FUNCTION_BLOCK _TcVnSize2_REAL_TestSuite EXTENDS TcUnit.FB_TestSuite
VAR
END_VAR

TestAddress();
TestClearReference();
TestClone();
TestTypeNameReturnsExpected();
TestIdentifierReturnsExpected();
//TestMakeReferenceToFollowsReference();
//TestMakeReferenceToUpdatesReference();
TestSize();
TestValueReturnsExpectedAfterInit();
TestValueReturnsExpectedAfterChange();
//TestSerializeTypeWith();
TestSerializeWith();
//TestTryDeserializeFrom();
//TestTryMakeReferenceToFollowsReference();
//TestTryMakeReferenceToUpdatesReference();

METHOD PUBLIC TestAddress
VAR
    _type : _TcVnSize2_REAL;
    notExpected : PVOID := 0;
    actual : PVOID;
END_VAR
TEST('TestAddress');

actual := _type.Address;

AssertFalse(
    Condition := (notExpected = actual),
    Message := 'Type did not return a valid address.'
);

TEST_FINISHED();
END_METHOD

METHOD PUBLIC TestClearReference
VAR
    _type : _ETcVn2dCodeSearchStrategy(ETcVn2dCodeSearchStrategy.TCVN_CSS_DEFAULT);
	target : ETcVn2dCodeSearchStrategy := ETcVn2dCodeSearchStrategy.TCVN_CSS_DEFAULT;
    expected : ETcVn2dCodeSearchStrategy := ETcVn2dCodeSearchStrategy.TCVN_CSS_DEFAULT;
    actual : ETcVn2dCodeSearchStrategy;
END_VAR
TEST('TestClearReference');

_type.MakeReferenceTo(target);
_type.ClearReference();
target := ETcVn2dCodeSearchStrategy.TCVN_CSS_FIRST_FLIPPED;

actual := _type.Value;

AssertEquals(
    Expected := expected,
    Actual := actual,
    Message := 'Value continued to follow target.'
);

TEST_FINISHED();
END_METHOD

METHOD PUBLIC TestClone
VAR
    _type : _TcVnSize2_REAL;
	clone : I_Datatype;
	isValidClone : BOOL;
	compareResult : DINT;
END_VAR
TEST('TestClone');

clone := _type.Clone();

isValidClone := clone <> 0;

IF isValidClone THEN
	compareResult := memcmp(_type.Address, clone.Address, clone.Size);
END_IF

AssertTrue(
	Condition := isValidClone,
	Message := 'Clone did not produce a clone'
);

AssertEquals_DINT(
	Expected := 0,
    Actual := compareResult,
    Message := 'Clone did not return a valid clone.'
);

clone.Dispose();

TEST_FINISHED();
END_METHOD

METHOD PUBLIC TestIdentifierReturnsExpected
VAR
    _type : _TcVnSize2_REAL;
    expected : STRING := 'TcVnSize2_REAL';
    actual : STRING;
END_VAR
TEST('TestIdentifierReturnsExpected');

actual := _type.Identifier;

AssertEquals_STRING(
    Expected := expected,
    Actual := actual,
    Message := 'Type did not return correct iec type.'
);

TEST_FINISHED();
END_METHOD

METHOD PUBLIC TestMakeReferenceToFollowsReference
VAR
    _type : _TcVnSize2_REAL;
	target : TcVnSize2_REAL;
    expected : TcVnSize2_REAL := (fWidth := 1.23, fHeight := 4.56);
    actual : TcVnSize2_REAL;
END_VAR
TEST('TestMakeReferenceToFollowsReference');

_type.MakeReferenceTo(target);
target.fWidth := 1.23;
target.fHeight := 4.56;

actual := _type.Value;

AssertEquals(
    Expected := expected,
    Actual := actual,
    Message := 'Value did not follow target change.'
);

TEST_FINISHED();
END_METHOD

METHOD PUBLIC TestMakeReferenceToUpdatesReference
VAR
    _type : _ETcVn2dCodeSearchStrategy(ETcVn2dCodeSearchStrategy.TCVN_CSS_DEFAULT);
	target : ETcVn2dCodeSearchStrategy := ETcVn2dCodeSearchStrategy.TCVN_CSS_DEFAULT;
    expected : ETcVn2dCodeSearchStrategy := ETcVn2dCodeSearchStrategy.TCVN_CSS_FIRST_FLIPPED;
    actual : ETcVn2dCodeSearchStrategy;
END_VAR
TEST('TestMakeReferenceToUpdatesReference');

_type.MakeReferenceTo(target);
_type.Value := ETcVn2dCodeSearchStrategy.TCVN_CSS_FIRST_FLIPPED;

actual := target;

AssertEquals(
    Expected := expected,
    Actual := actual,
    Message := 'Value did not update target.'
);

TEST_FINISHED();
END_METHOD

METHOD PUBLIC TestSerializeTypeWith
VAR
    _type : _TcVnSize2_REAL;
    serializer : JsonSerializer;
    //expected : STRING(500) := '{"typeName":"STRUCT","identifier":"TcVnSize2_REAL","members":{"fWidth":{"typeName":"REAL","minValue":-3.4028230607370967e38,"maxValue":3.4028230607370967      }';
    expected : STRING(500) := '';
    actual : STRING(500);
END_VAR
TEST('TestSerializeTypeWith');

serializer.Reset();
_type.SerializeTypeWith(serializer);
serializer.TryGetSerializedData(ADR(actual), SIZEOF(actual));

AssertEquals_STRING(
    Expected := expected,
    Actual := actual,
    Message := 'Serialization of type did not return correct string.'
);

TEST_FINISHED();
END_METHOD

METHOD PUBLIC TestSerializeWith
VAR
    _type : _TcVnSize2_REAL;
    serializer : JsonSerializer;
    expected : STRING := '{"fWidth":0.0,"fHeight":0.0}';
    actual : STRING(500);
END_VAR
TEST('TestSerializeWith');

serializer.Reset();
_type.SerializeWith(serializer);
serializer.TryGetSerializedData(ADR(actual), SIZEOF(actual));

AssertEquals_STRING(
    Expected := expected,
    Actual := actual,
    Message := 'Serialization of type data did not return correct string.'
);

TEST_FINISHED();
END_METHOD

METHOD PUBLIC TestSize
VAR
    _type : _TcVnSize2_REAL;
    expected : UDINT := SIZEOF(TcVnSize2_REAL);
    actual : UDINT;
END_VAR
TEST('TestSize');

actual := _type.Size;

AssertEquals_UDINT(
    Expected := Expected,
    Actual := actual,
    Message := 'Type did not return the correct size.'
);

TEST_FINISHED();
END_METHOD

METHOD PUBLIC TestTryDeserializeFrom
VAR
    deserializer : JsonDeserializer;
    feedback : DeserializerFeedback;
    json : STRING := '"TCVN_CSS_DEFAULT"';
    _type : _ETcVn2dCodeSearchStrategy(ETcVn2dCodeSearchStrategy.TCVN_CSS_DEFAULT);
    expected : ETcVn2dCodeSearchStrategy := ETcVn2dCodeSearchStrategy.TCVN_CSS_DEFAULT;
    actual : ETcVn2dCodeSearchStrategy;
 END_VAR
TEST('TestTryDeserializeFrom');

deserializer.Reset();
deserializer.TryLoad(json);
_type.TryDeserializeFrom(Deserializer, Feedback);

actual := _type.Value;

AssertEquals(
    Expected := expected,
    Actual := actual,
    Message := 'Type did not deserialize correctly.'
);

TEST_FINISHED();
END_METHOD

METHOD PUBLIC TestTryMakeReferenceToFollowsReference
VAR
    _type : _TcVnSize2_REAL;
	target : _TcVnSize2_REAL;
    expected : TcVnSize2_REAL := (fWidth := 1.23, fHeight := 4.56);
    actual : TcVnSize2_REAL;
END_VAR
TEST('TestTryMakeReferenceToFollowsReference');

_type.TryMakeReferenceTo(target);
target.Value.fHeight := 1.23;
target.Value.fHeight := 4.56;

actual := _type.Value;

AssertEquals(
    Expected := expected,
    Actual := actual,
    Message := 'Value did not follow target change.'
);

TEST_FINISHED();
END_METHOD

METHOD PUBLIC TestTryMakeReferenceToUpdatesReference
VAR
    _type : _ETcVn2dCodeSearchStrategy(ETcVn2dCodeSearchStrategy.TCVN_CSS_DEFAULT);
	target : _ETcVn2dCodeSearchStrategy(ETcVn2dCodeSearchStrategy.TCVN_CSS_DEFAULT);
    expected : ETcVn2dCodeSearchStrategy := ETcVn2dCodeSearchStrategy.TCVN_CSS_FIRST_FLIPPED;
    actual : ETcVn2dCodeSearchStrategy;
END_VAR
TEST('TestTryMakeReferenceToUpdatesReference');

_type.TryMakeReferenceTo(target);
_type.Value := ETcVn2dCodeSearchStrategy.TCVN_CSS_FIRST_FLIPPED;

actual := target.Value;

AssertEquals(
    Expected := expected,
    Actual := actual,
    Message := 'Value did not update target.'
);

TEST_FINISHED();
END_METHOD

METHOD PUBLIC TestTypeNameReturnsExpected
VAR
    _type : _TcVnSize2_REAL;
    expected : STRING := 'STRUCT';
    actual : STRING;
END_VAR
TEST('TestTypeNameReturnsExpected');

actual := _type.TypeName;

AssertEquals_STRING(
    Expected := expected,
    Actual := actual,
    Message := 'Type did not return correct iec type.'
);

TEST_FINISHED();
END_METHOD

METHOD PUBLIC TestValueReturnsExpectedAfterChange
VAR
    _type : _TcVnSize2_REAL;
    expected : TcVnSize2_REAL := (fWidth := 1.23, fHeight := 4.56);
    actual : TcVnSize2_REAL;
END_VAR
TEST('TestValueReturnsExpectedAfterChange');

_type.Value.fWidth := 1.23;
_type.Value.fHeight := 4.56;

actual := _type.Value;

AssertEquals(
    Expected := expected,
    Actual := actual,
    Message := 'Expected value not returned after change.'
);

TEST_FINISHED();
END_METHOD

METHOD PUBLIC TestValueReturnsExpectedAfterInit
VAR
    _type : _TcVnSize2_REAL;
    expected : TcVnSize2_REAL;
    actual : TcVnSize2_REAL;
END_VAR
TEST('TestValueReturnsExpectedAfterInit');

actual := _type.Value;

AssertEquals(
    Expected := expected,
    Actual := actual,
    Message := 'Expected value not returned after Init.'
);

TEST_FINISHED();
END_METHOD

END_FUNCTION_BLOCK

(* stored: Version 1.1.0.1, ProductVersion 3.1.4024.13
   POU _TcVnSize2_REAL_TestSuite: Id {6ff71fa2-be53-0011-2c7a-27a055ca06e0}, SpecialFunc None
   Method TestAddress: Id {f7467aa7-aae7-08b6-157c-a10b3c1360b7}
   Method TestClearReference: Id {e1cd17b4-ab29-094f-33e7-5372884badd8}
   Method TestClone: Id {25d92291-f963-09b5-03c3-579e655d3aee}
   Method TestIdentifierReturnsExpected: Id {9c0e1868-06c2-0429-191a-68dd437caaaf}
   Method TestMakeReferenceToFollowsReference: Id {0637c88c-9984-08cf-2c97-55a639117630}
   Method TestMakeReferenceToUpdatesReference: Id {8c989be6-3d37-099c-0ee3-8e3accd838ff}
   Method TestSerializeTypeWith: Id {12581887-c612-004b-1c0c-77a836dea60f}
   Method TestSerializeWith: Id {18d379cb-fe6a-06c5-09c7-93916a866403}
   Method TestSize: Id {51752e32-4256-0e77-2399-e9016d2bcb53}
   Method TestTryDeserializeFrom: Id {d4245a37-da6f-0573-1f05-eff2c86969a7}
   Method TestTryMakeReferenceToFollowsReference: Id {bc2b41dc-f854-01f5-26fb-9c113f7ed814}
   Method TestTryMakeReferenceToUpdatesReference: Id {3d35944a-9f91-0c0e-008e-42cfb0b5ebe7}
   Method TestTypeNameReturnsExpected: Id {46d3f455-f7d8-0b81-1f28-28ac203229c0}
   Method TestValueReturnsExpectedAfterChange: Id {6ead7160-69a3-086e-3d5b-ff163d04cb7b}
   Method TestValueReturnsExpectedAfterInit: Id {69cd22c8-7445-0184-0e89-7c649cbebafd} *)
